Fanuc KAREL source: ADD_REALPC.kl

PROGRAM T
%NOLOCKGROUP
VAR
 v0 : ARRAY[20] OF BYTE
 v1 : INTEGER
 v2 : REAL
 v3 : INTEGER
BEGIN
 ADD_REALPC(v0, v1, v2, v3)
END T
